Staubli VAL3: MainKey.pgx

program MainKey(num x_nKey)
  local num l_nKey
begin
  //
  switch x_nKey
    //
    case 271
      call OnF1()
    break
    //编辑
    case 272
      call OnF2()
    break
    //
    case 273
      //call OnF3()
    break
    //
    case 274
      // call OnF4()
    break
    //
    case 275
    break
    //
    case 276
      //call OnF6()
    break
    //save
    case 277
      call OnF7()
    break
    //返回
    case 278
      call OnF8("是否返回")
    break

  endSwitch
end
